{attribute 'qualified_only'}
VAR_GLOBAL
	AxisX_Inputs		: AxisInputs;
	AxisY_Inputs		: AxisInputs;
	AxisZ_Inputs		: AxisInputs;
END_VAR

(* stored: Version 1.1.0.1, ProductVersion 3.1.4024.10
   GVL Inputs: Id {c055cae3-14d0-40ee-9f1f-7b5ae4d4b8e4} *)
